{attribute 'GeneratedUsingTerminal: EP2816-0008-0019'}
{attribute addProperty BoxType "EP2816-0008-0019"}
{attribute addProperty Description "EP2816-0008 16 Ch. Dig. Output 24V, 0,5A, Diagnostic, D-SUB25"}
{attribute addProperty Physics "YY"}
{attribute addProperty Id "DIG_Diag_Inputs_Channel_1AT %I*DIG_Diag_Inputs_Channel_584303BF8DIG_Diag_Inputs_Channel_2AT %I*DIG_Diag_Inputs_Channel_584303BF8DIG_Inputs_DeviceAT %I*DIG_Inputs_Device_E94E5BF95DIG_Outputs_Channel_1AT %Q*DIG_Outputs_Channel_28AC1A9E8DIG_Outputs_Channel_2AT %Q*DIG_Outputs_Channel_28AC1A9E8DIG_Outputs_DeviceAT %Q*DIG_Outputs_Device_36A5EF172WcStateAT %I*WcState_9091E0EB2InfoDataAT %I*InfoData_32EB74EA10"}
{attribute addProperty CRC "19489865"}
{attribute addProperty Size "51"}
TYPE EP2816_01296449 EXTENDS EtcSlaveBoxBase_77A0E4A7 :
STRUCT
	{attribute addProperty Name "DIG_Diag_Inputs_Channel_1"}
	DIG_Diag_Inputs_Channel_1 : DIG_Diag_Inputs_Channel_584303BF;
	{attribute addProperty Name "DIG_Diag_Inputs_Channel_2"}
	DIG_Diag_Inputs_Channel_2 : DIG_Diag_Inputs_Channel_584303BF;
	{attribute addProperty Name "DIG_Inputs_Device"}
	DIG_Inputs_Device : DIG_Inputs_Device_E94E5BF9;
	{attribute addProperty Name "DIG_Outputs_Channel_1"}
	DIG_Outputs_Channel_1 : DIG_Outputs_Channel_28AC1A9E;
	{attribute addProperty Name "DIG_Outputs_Channel_2"}
	DIG_Outputs_Channel_2 : DIG_Outputs_Channel_28AC1A9E;
	{attribute addProperty Name "DIG_Outputs_Device"}
	DIG_Outputs_Device : DIG_Outputs_Device_36A5EF17;
	{attribute addProperty Name "WcState"}
	WcState : WcState_9091E0EB;
	{attribute addProperty Name "InfoData"}
	InfoData : InfoData_32EB74EA;
END_STRUCT
END_TYPE

(* stored: Version 1.2.0.0, ProductVersion 3.1.4024.9
   DUT EP2816_01296449: Id {63749724-c75b-48b9-be7a-17ec9857112e} *)
